(* CoDeSys 2.3.5.6 project: lyjak_02.pro *)
(* Libraries: Standard.lib 4.1.15 17:23:13, SYSLIBCALLBACK.LIB 4.1.15 17:23:13 *)

(* PLC configuration (modules and I/O channels)
Local I/O [EC4P_LocalIO] node 0, in %IB0 out %QB0 {EC4P_LocalInt = 0}
  I1 AT %IX0.0 [LocalBitInput] Input I1
  I2 AT %IX0.1 [LocalBitInput] Input I2
  I3 AT %IX0.2 [LocalBitInput] Input I3
  I4 AT %IX0.3 [LocalBitInput] Input I4
  I5 AT %IX0.4 [LocalBitInput] Input I5
  I6 AT %IX0.5 [LocalBitInput] Input I6
  I7 AT %IX0.6 [LocalBitInput] Input I7
  I8 AT %IX0.7 [LocalBitInput] Input I8
  I9 AT %IX1.0 [LocalBitInput] Input I9
  I10 AT %IX1.1 [LocalBitInput] Input I10
  I11 AT %IX1.2 [LocalBitInput] Input I11
  I12 AT %IX1.3 [LocalBitInput] Input I12
  I13 AT %IX1.4 [LocalDiagInput] Diagnostic Input I13
  I14 AT %IX1.5 [LocalDiagInput] Diagnostic Input I14
  I15 AT %IX1.6 [LocalDiagInput] Diagnostic Input I15
  I16 AT %IX1.7 [LocalDiagInput] Diagnostic Input I16
  I7_Analog AT %IW2 [LocalAnalogIn] Input I7, 10Bit, 0-10VDC
  I8_Analog AT %IW4 [LocalAnalogIn] Input I8, 10Bit, 0-10VDC
  I11_Analog AT %IW6 [LocalAnalogIn] Input I11, 10Bit, 0-10VDC
  I12_Analog AT %IW8 [LocalAnalogIn] Input I12, 10Bit, 0-10VDC
  Transistor Outputs [EC4P_TOutputs] node 0, in %IB10 out %QB0
    Q1 AT %QX0.0 [LocalBitOutput] Transistor-Output Q1
    Q2 AT %QX0.1 [LocalBitOutput] Transistor-Output Q2
    Q3 AT %QX0.2 [LocalBitOutput] Transistor-Output Q3
    Q4 AT %QX0.3 [LocalBitOutput] Transistor-Output Q4
    Q5 AT %QX0.4 [LocalBitOutput] Transistor-Output Q5
    Q6 AT %QX0.5 [LocalBitOutput] Transistor-Output Q6
    Q7 AT %QX0.6 [LocalBitOutput] Transistor-Output Q7
    Q8 AT %QX0.7 [LocalBitOutput] Transistor-Output Q8
  No Analog Output [EC4P_NoAnalogOutput] node 1, in %IB10 out %QB1
  No Keys [EC4P_NoKeys] node 2, in %IB10 out %QB1
  No Counter [EC4P_NoCounter] node 3, in %IB10 out %QB1
Extension [EC4P_Extension] node 1, in %IB10 out %QB1
  No Extension [EC4P_NoExtension] node 0, in %IB10 out %QB1
*)

(* POU PLC_PRG, CFC *)
PROGRAM PLC_PRG
VAR
	TP1: TP;
	TP2: TP;
	ON: BOOL;
	TTP1: TIME;
	FTRIG1: F_TRIG;
	TTP2: TIME;
	RTRIG1: R_TRIG;
	TP3: TP;
	TP4: TP;
	FTRIG2: F_TRIG;
	TTP3: TIME;
	TTP4: TIME;
END_VAR
VAR (* helpers for the ST form of the networks *)
	_t35 : BOOL;
	_t37 : BOOL;
	_t32 : BOOL;
	_t11 : BOOL;
	_t12 : BOOL;
	_t10 : BOOL;
	_t58 : BOOL;
	_t53 : BOOL;
	_t183 : BOOL;
	_t185 : BOOL;
	_t38 : BOOL;
	_t39 : BOOL;
	_t174 : BOOL;
	_t61 : BOOL;
	_t164 : BOOL;
	_t187 : BOOL;
	_t188 : BOOL;
	_t257 : BOOL;
	_t267 : BOOL;
	_t305 : BOOL;
	_t276 : BOOL;
	_t273 : BOOL;
	_t277 : BOOL;
	_t290 : BOOL;
	_t289 : BOOL;
	_t300 : BOOL;
	_t299 : BOOL;
	_t306 : BOOL;
	_t315 : BOOL;
	_t314 : BOOL;
	_t346 : BOOL;
	_t333 : BOOL;
	_t332 : BOOL;
END_VAR
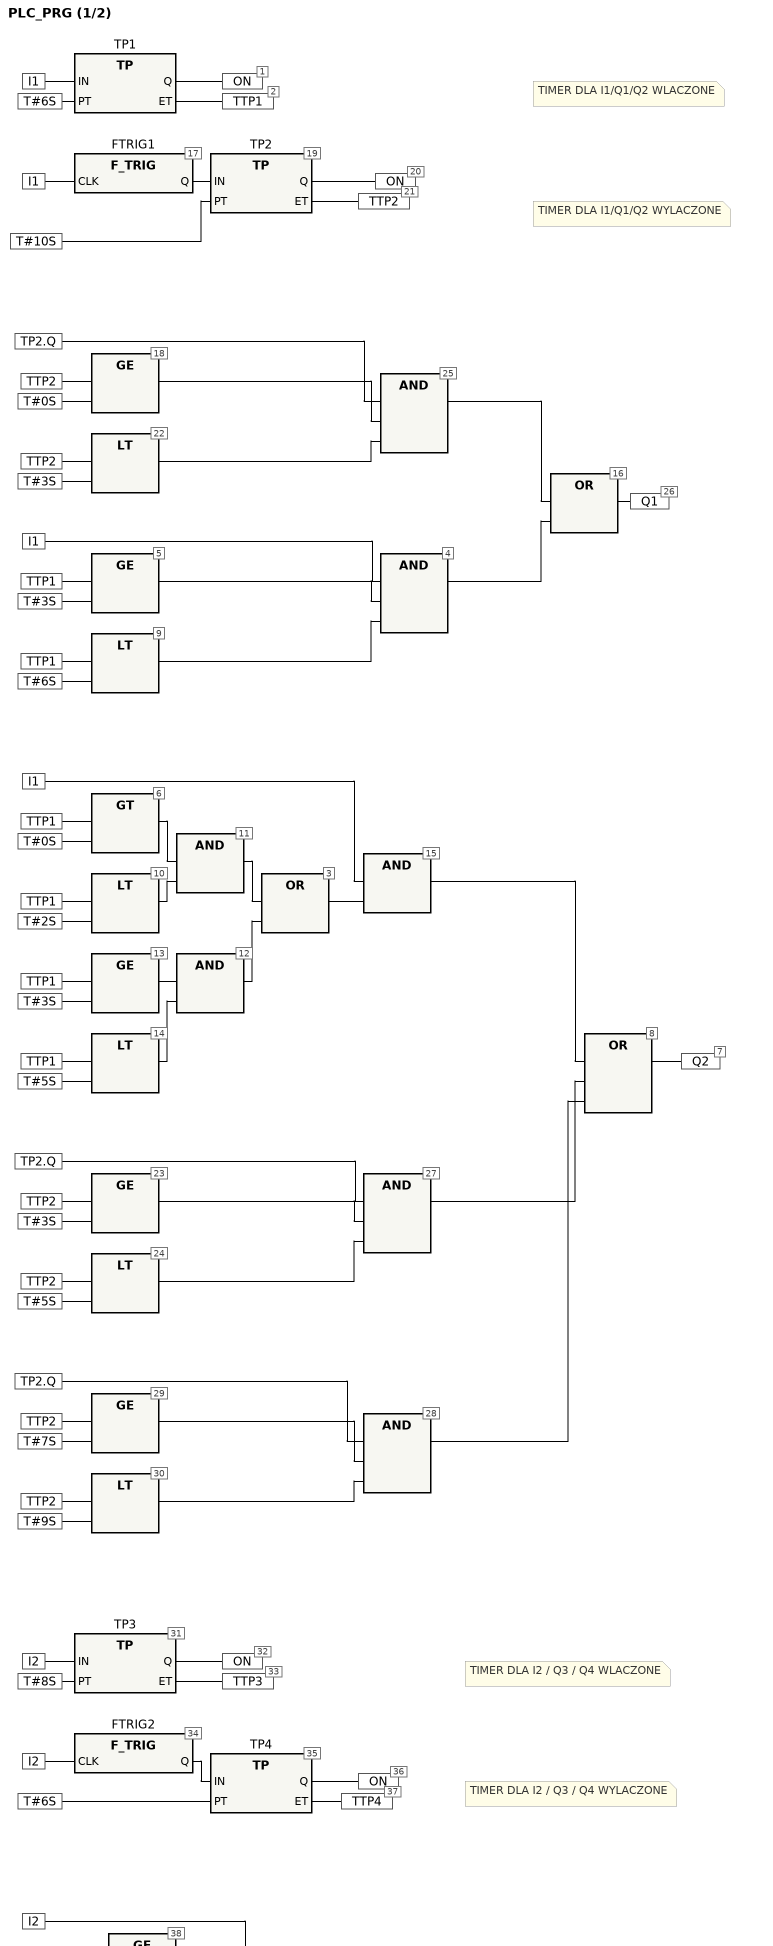
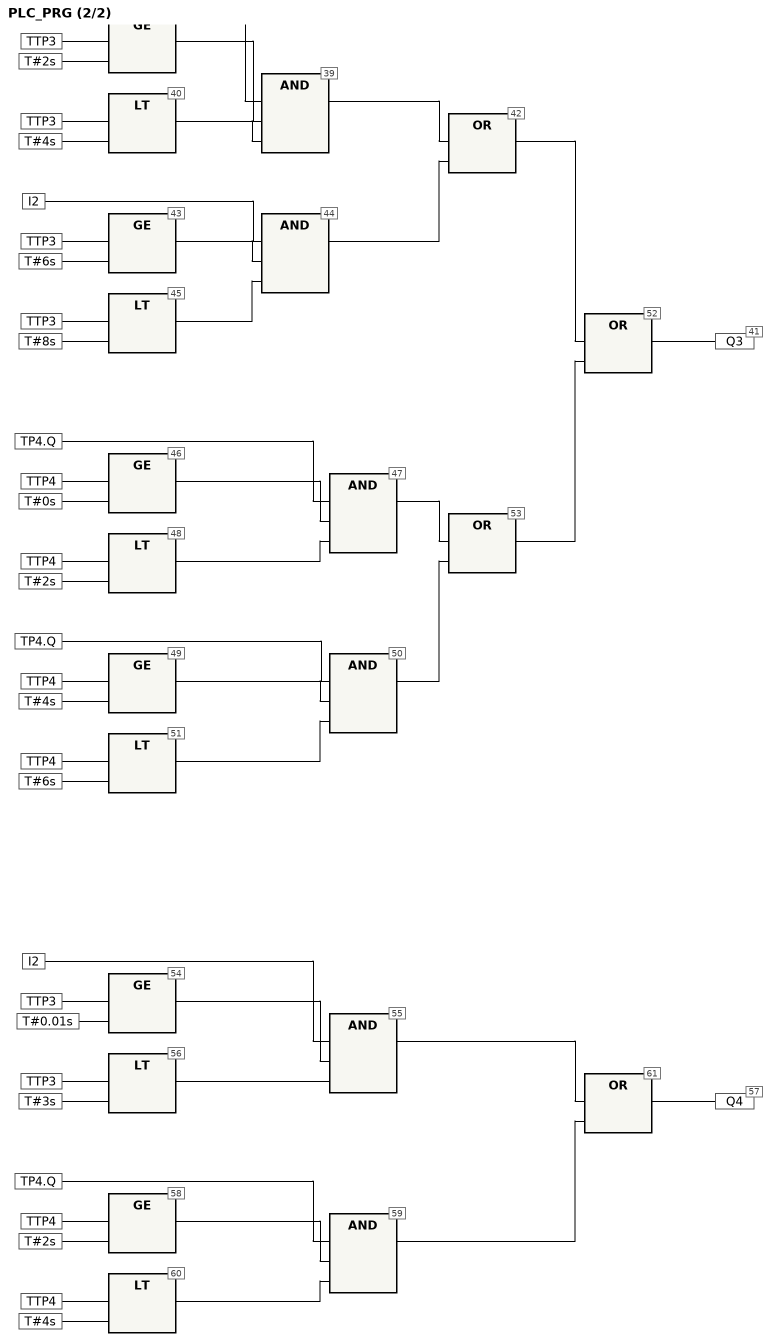
_CFC_ (* Continuous Function Chart, elements in execution order *)
#0 TP1:TP(IN: I1, PT: T#6S)
#1 ON <= #0.Q
#2 TTP1 <= #0.ET
#3 OR(#11, #12)
#4 AND(I1, #5, #9)
#5 GE(TTP1, T#3S)
#6 GT(TTP1, T#0S)
#7 Q2 <= #8
#8 OR(#15, #27, #28)
#9 LT(TTP1, T#6S)
#10 LT(TTP1, T#2S)
#11 AND(#6, #10)
#12 AND(#13, #14)
#13 GE(TTP1, T#3S)
#14 LT(TTP1, T#5S)
#15 AND(I1, #3)
#16 OR(#25, #4)
#17 FTRIG1:F_TRIG(CLK: I1)
#18 GE(TTP2, T#0S)
#19 TP2:TP(IN: #17.Q, PT: T#10S)
#20 ON <= #19.Q
#21 TTP2 <= #19.ET
#22 LT(TTP2, T#3S)
#23 GE(TTP2, T#3S)
#24 LT(TTP2, T#5S)
#25 AND(TP2.Q, #18, #22)
#26 Q1 <= #16
#27 AND(TP2.Q, #23, #24)
#28 AND(TP2.Q, #29, #30)
#29 GE(TTP2, T#7S)
#30 LT(TTP2, T#9S)
(* TIMER DLA I1/Q1/Q2 WYLACZONE *)
(* TIMER DLA I1/Q1/Q2 WLACZONE *)
#31 TP3:TP(IN: I2, PT: T#8S)
#32 ON <= #31.Q
#33 TTP3 <= #31.ET
#34 FTRIG2:F_TRIG(CLK: I2)
#35 TP4:TP(IN: #34.Q, PT: T#6S)
#36 ON <= #35.Q
#37 TTP4 <= #35.ET
(* TIMER DLA I2 / Q3 / Q4 WYLACZONE *)
(* TIMER DLA I2 / Q3 / Q4 WLACZONE *)
#38 GE(TTP3, T#2s)
#39 AND(I2, #38, #40)
#40 LT(TTP3, T#4s)
#41 Q3 <= #52
#42 OR(#39, #44)
#43 GE(TTP3, T#6s)
#44 AND(I2, #43, #45)
#45 LT(TTP3, T#8s)
#46 GE(TTP4, T#0s)
#47 AND(TP4.Q, #46, #48)
#48 LT(TTP4, T#2s)
#49 GE(TTP4, T#4s)
#50 AND(TP4.Q, #49, #51)
#51 LT(TTP4, T#6s)
#52 OR(#42, #53)
#53 OR(#47, #50)
#54 GE(TTP3, T#0.01s)
#55 AND(I2, #54, #56)
#56 LT(TTP3, T#3s)
#57 Q4 <= #61
#58 GE(TTP4, T#2s)
#59 AND(TP4.Q, #58, #60)
#60 LT(TTP4, T#4s)
#61 OR(#55, #59)
_END_CFC_
(* the same logic as Structured Text *)
TP1(IN := I1, PT := T#6S);
ON := TP1.Q;
TTP1 := TP1.ET;
_t32 := _t35 OR _t37;
_t10 := I1 AND _t11 AND _t12;
_t11 := TTP1 >= T#3S;
Q2 := _t58;
_t58 := _t53 OR _t183 OR _t185;
_t12 := TTP1 < T#6S;
_t35 := (TTP1 > T#0S) AND (TTP1 < T#2S);
_t37 := _t38 AND _t39;
_t38 := TTP1 >= T#3S;
_t39 := TTP1 < T#5S;
_t53 := I1 AND _t32;
_t61 := _t174 OR _t10;
FTRIG1(CLK := I1);
_t164 := TTP2 >= T#0S;
TP2(IN := FTRIG1.Q, PT := T#10S);
ON := TP2.Q;
TTP2 := TP2.ET;
_t174 := TP2.Q AND _t164 AND (TTP2 < T#3S);
Q1 := _t61;
_t183 := TP2.Q AND (TTP2 >= T#3S) AND (TTP2 < T#5S);
_t185 := TP2.Q AND _t187 AND _t188;
_t187 := TTP2 >= T#7S;
_t188 := TTP2 < T#9S;
(* TIMER DLA I1/Q1/Q2 WYLACZONE *)
(* TIMER DLA I1/Q1/Q2 WLACZONE *)
TP3(IN := I2, PT := T#8S);
ON := TP3.Q;
TTP3 := TP3.ET;
FTRIG2(CLK := I2);
TP4(IN := FTRIG2.Q, PT := T#6S);
ON := TP4.Q;
TTP4 := TP4.ET;
(* TIMER DLA I2 / Q3 / Q4 WYLACZONE *)
(* TIMER DLA I2 / Q3 / Q4 WLACZONE *)
_t267 := I2 AND (TTP3 >= T#2s) AND _t257;
_t257 := TTP3 < T#4s;
Q3 := _t305;
_t273 := _t267 OR _t276;
_t276 := I2 AND (TTP3 >= T#6s) AND _t277;
_t277 := TTP3 < T#8s;
_t289 := TP4.Q AND (TTP4 >= T#0s) AND _t290;
_t290 := TTP4 < T#2s;
_t299 := TP4.Q AND (TTP4 >= T#4s) AND _t300;
_t300 := TTP4 < T#6s;
_t305 := _t273 OR _t306;
_t306 := _t289 OR _t299;
_t314 := I2 AND (TTP3 >= T#0.01s) AND _t315;
_t315 := TTP3 < T#3s;
Q4 := _t346;
_t332 := TP4.Q AND (TTP4 >= T#2s) AND _t333;
_t333 := TTP4 < T#4s;
_t346 := _t314 OR _t332;
END_PROGRAM
